(* IEC 61131-3 sources: ax-factoryio-assembler/src/ControlModules/TwoAxisPickPlace, 2 files *)

(* ---- States.st ---- *)
USING System.Timer;

NAMESPACE Demo.ControlModule.States.TwoAxisPickPlace

INTERFACE IPickPlaceState
    METHOD Start END_METHOD
    METHOD Reset END_METHOD
    METHOD Stop END_METHOD
    METHOD EmergencyStop END_METHOD
    METHOD Cycle END_METHOD
    METHOD OnEntry END_METHOD
    METHOD OnExit END_METHOD
    METHOD GetStateName:STRING END_METHOD
END_INTERFACE

CLASS StateBase IMPLEMENTS IPickPlaceState
    VAR PUBLIC
        Device: REF_TO TwoAxisPickPlace;
        NextState: IPickPlaceState;
        Name: STRING;
    END_VAR

    METHOD PUBLIC Start
        ;
    END_METHOD

    METHOD PUBLIC Reset
        ;
    END_METHOD

    METHOD PUBLIC Stop
        ;
    END_METHOD

    METHOD PUBLIC Cycle
        ;
    END_METHOD

    METHOD PUBLIC OnEntry
        ;
    END_METHOD

    METHOD PUBLIC IsDone:BOOL
        IsDone := FALSE;
    END_METHOD

    METHOD PUBLIC EmergencyStop
        ;
    END_METHOD

    METHOD PUBLIC OnExit
        ;
    END_METHOD

    METHOD PUBLIC GetStateName : STRING
        GetStateName := Name;
    END_METHOD
END_CLASS

CLASS IdleState EXTENDS StateBase
    METHOD PUBLIC OVERRIDE Start
        Device^.IsDone := FALSE;
        Device^.SetState(NextState);
    END_METHOD
END_CLASS

CLASS StartingState EXTENDS StateBase
    METHOD PUBLIC OVERRIDE Cycle
        Device^.MoveZ^ := TRUE;
        Device^.SetState(NextState);
    END_METHOD
END_CLASS

CLASS PickMovingZDownState EXTENDS StateBase
    VAR PRIVATE
        _delayTimer: OnDelay;
    END_VAR

    METHOD PUBLIC OVERRIDE OnEntry
        _delayTimer(FALSE);
    END_METHOD

    METHOD PUBLIC OVERRIDE Cycle
        _delayTimer(NOT (Device^.MovingZ^), LT#200ms);
        IF _delayTimer.output THEN
            Device^.Grab^ := TRUE;
            Device^.SetState(NextState);
        END_IF;
    END_METHOD
END_CLASS

CLASS GrabbingState EXTENDS StateBase
    VAR PRIVATE
        _delayTimer: OnDelay;
    END_VAR

    METHOD PUBLIC OVERRIDE OnEntry
        _delayTimer(FALSE);
    END_METHOD

    METHOD PUBLIC OVERRIDE Cycle
        _delayTimer(Device^.ItemDetected^, LT#200ms);
        IF _delayTimer.output THEN
            Device^.MoveZ^ := FALSE;
            Device^.SetState(NextState);
        END_IF;
    END_METHOD
END_CLASS

CLASS PickMovingZUpState EXTENDS StateBase
    VAR PRIVATE
        _delayTimer: OnDelay;
    END_VAR

    METHOD PUBLIC OVERRIDE OnEntry
        _delayTimer(FALSE);
    END_METHOD

    METHOD PUBLIC OVERRIDE Cycle
        _delayTimer(NOT (Device^.MovingZ^), LT#200ms);
        IF _delayTimer.output THEN
            Device^.MoveX^ := TRUE;
            Device^.SetState(NextState);
        END_IF;
    END_METHOD
END_CLASS

CLASS MovingXRightState EXTENDS StateBase
    VAR PRIVATE
        _delayTimer: OnDelay;
    END_VAR

    METHOD PUBLIC OVERRIDE OnEntry
        _delayTimer(FALSE);
    END_METHOD

    METHOD PUBLIC OVERRIDE Cycle
        _delayTimer(NOT (Device^.MovingX^), LT#200ms);
        IF _delayTimer.output THEN
            Device^.MoveZ^ := TRUE;
            Device^.SetState(NextState);
        END_IF;
    END_METHOD
END_CLASS

Class PlaceMovingZDownState EXTENDS StateBase
    VAR PRIVATE
        _delayTimer: OnDelay;
    END_VAR

    METHOD PUBLIC OVERRIDE OnEntry
        _delayTimer(FALSE);
    END_METHOD

    METHOD PUBLIC OVERRIDE Cycle
        _delayTimer(NOT (Device^.MovingZ^), LT#200ms);
        IF _delayTimer.output THEN
            Device^.MoveZ^:=FALSE;
            Device^.Grab^:=FALSE;
            Device^.SetState(NextState);
        END_IF;
    END_METHOD
END_CLASS

CLASS PlaceMovingZUpState EXTENDS StateBase
    VAR PRIVATE
        _delayTimer: OnDelay;
    END_VAR

    METHOD PUBLIC OVERRIDE OnEntry
        _delayTimer(FALSE);
    END_METHOD

    METHOD PUBLIC OVERRIDE Cycle
        Device^.MoveZ^:=FALSE;

        _delayTimer(NOT (Device^.MovingZ^), LT#200ms);
        IF _delayTimer.output THEN
            Device^.SetState(NextState);
        END_IF;
    END_METHOD
END_CLASS

CLASS CompleteState EXTENDS StateBase
    METHOD PUBLIC OVERRIDE Cycle
        Device^.IsDone := TRUE;
        Device^.MoveZ^:=FALSE;
        Device^.MoveX^:=FALSE;
        Device^.Grab^:=FALSE;
        Device^.SetState(NextState);
    END_METHOD
END_CLASS

CLASS StopState EXTENDS StateBase
    METHOD PUBLIC OVERRIDE Reset
        Device^.SetState(NextState);
    END_METHOD
END_CLASS

CLASS ResetingState EXTENDS StateBase
    METHOD PUBLIC OVERRIDE OnEntry
        Device^.MoveZ^:=FALSE;
        Device^.MoveX^:=FALSE;
        Device^.Grab^:=FALSE;
        Device^.IsDone := FALSE;
    END_METHOD

    METHOD PUBLIC OVERRIDE Cycle
        Device^.SetState(NextState);
    END_METHOD
END_CLASS

CLASS EmergencyStopState EXTENDS StateBase
    METHOD PUBLIC OVERRIDE Reset
        Device^.SetState(NextState);
    END_METHOD
END_CLASS

END_NAMESPACE

(* ---- TwoAxisPickPlace.st ---- *)
USING Demo.ControlModule.States.TwoAxisPickPlace;
USING System.Timer;

NAMESPACE Demo.ControlModule

INTERFACE ITwoAxisPickPlace EXTENDS ICyclic
        METHOD Init
        END_METHOD

        METHOD SetState
            VAR_INPUT
                state : IPickPlaceState;
            END_VAR
        END_METHOD

        METHOD GetStateName : STRING
        END_METHOD

        METHOD Start
        END_METHOD

        METHOD Reset END_METHOD

        METHOD Stop END_METHOD

        METHOD EmergencyStop END_METHOD

        METHOD GetIsDone:BOOL END_METHOD
END_INTERFACE

CLASS TwoAxisPickPlace IMPLEMENTS ITwoAxisPickPlace
    VAR PUBLIC
        MovingX : REF_TO BOOL;
        MovingZ: REF_TO BOOL;
        ItemDetected : REF_TO BOOL;

        MoveX: REF_TO BOOL;
        MoveZ: REF_TO BOOL;
        Grab: REF_TO BOOL;
        InitState: IPickPlaceState;
        IsDone: BOOL;
        TheStopState: IPickPlaceState;
        TheResetState: IPickPlaceState;
    END_VAR

    VAR PRIVATE
        _status: IPickPlaceState;
    END_VAR

    METHOD PUBLIC Init
        _status := InitState;
    END_METHOD

    METHOD PUBLIC SetState
        VAR_INPUT
            state : IPickPlaceState;
        END_VAR
        _status.OnExit();
        _status := state;
        _status.OnEntry();
    END_METHOD

    METHOD PUBLIC GetStateName : STRING
        GetStateName:= _status.GetStateName();
    END_METHOD

    METHOD PUBLIC Start
        _status.Start();
    END_METHOD

    METHOD PUBLIC Reset
        _status.Reset();
    END_METHOD

    METHOD PUBLIC Stop
        This.SetState(TheStopState);
    END_METHOD

    METHOD PUBLIC EmergencyStop
        This.SetState(TheStopState);
    END_METHOD

    METHOD PUBLIC Cycle
        _status.Cycle();
    END_METHOD

    METHOD PUBLIC GetIsDone: BOOL
        GetIsDone := IsDone;
    END_METHOD
END_CLASS

END_NAMESPACE
